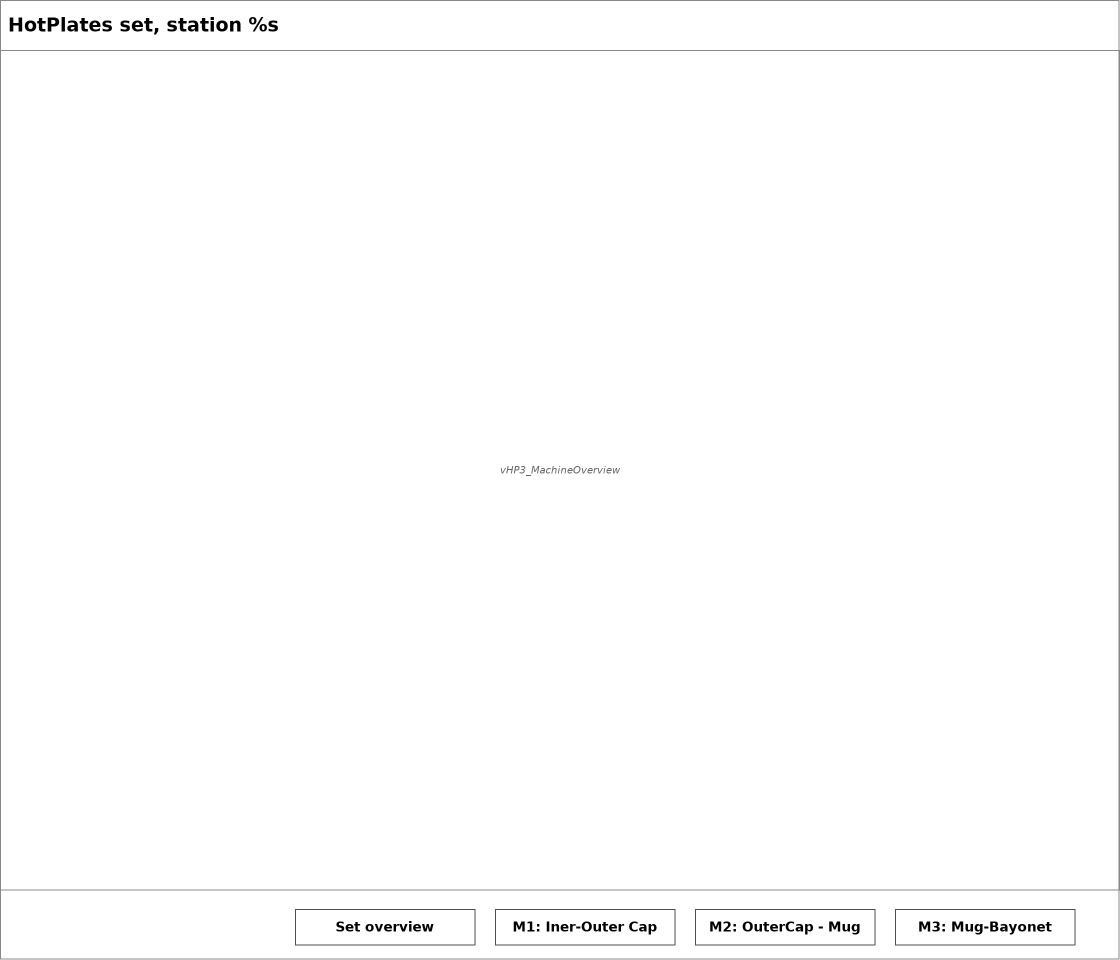
VISUALIZATION vHP3_MainSet  // 1120x960
VAR_IN_OUT
	fbHP_M1: fbHPv3_Control;
	fbHP_M2: fbHPv3_Control;
	fbHP_M3: fbHPv3_Control;
END_VAR
VAR_INPUT
	NestNumber: INT:= 1;
	sSocketName: STRING;	
END_VAR
VAR
	iButtonIndex: INT;
END_VAR
    Rectangle (0,890 1120x70), colour variable: GVL.adwHPNestsColorTable[NestNumber]
    Rectangle (0,0 1120x50), colour variable: GVL.adwHPNestsColorTable[NestNumber]
    Rectangle (295,909 180x36), "Set overview"
        OnMouseClick: FrameSelectionChange Selection=SelectedFrame=2d948332-6323-4ce4-b5f8-a8f9ee9afdb0, GlobSel=AssignType=Expression, SelType=Locally
        OnMouseClick: execute { iButtonIndex := 0; }
    Rectangle (495,909 180x36), "M1: Iner-Outer Cap"
        OnMouseClick: FrameSelectionChange Selection=SelectedFrame=2d948332-6323-4ce4-b5f8-a8f9ee9afdb0, Selection=1, GlobSel=AssignType=Expression, SelType=Locally
        OnMouseClick: execute { iButtonIndex := 1; }
    Rectangle (695,909 180x36), "M2: OuterCap - Mug"
        OnMouseClick: FrameSelectionChange Selection=SelectedFrame=2d948332-6323-4ce4-b5f8-a8f9ee9afdb0, Selection=2, GlobSel=AssignType=Expression, SelType=Locally
        OnMouseClick: execute { iButtonIndex := 2; }
    Rectangle (895,909 180x36), "M3: Mug-Bayonet"
        OnMouseClick: FrameSelectionChange Selection=SelectedFrame=2d948332-6323-4ce4-b5f8-a8f9ee9afdb0, Selection=3, GlobSel=AssignType=Expression, SelType=Locally
        OnMouseClick: execute { iButtonIndex := 3; }
    Frame (0,50 1120x840)
        shows vHP3_MachineOverview(fbHP_M1 := fbHP_M1, fbHP_M2 := fbHP_M2, fbHP_M3 := fbHP_M3)
        shows vHP3_MainMachine(fbHP := fbHP_M1)
        shows vHP3_MainMachine(fbHP := fbHP_M2)
        shows vHP3_MainMachine(fbHP := fbHP_M3)
    Rectangle (5,5 530x40), "HotPlates set, station %s", text variable: sSocketName, text list: 'tlHPv3', text index: 0
END_VISUALIZATION

(* stored: Version 1.1.0.1, ProductVersion 3.1.4024.13
   Visu vHP3_MainSet: Id {27965ebd-9d89-4f56-b668-4ab67e1c19c8} *)
